// TIA Portal V20 export
TYPE "typeCmHmiInterfaceSoftCam"
// stored: Access Published, Namespace Unit1.Em4
   STRUCT
      sideTapeFixStageAxisX : "Unit1.Em4.typeCmHmiInterfaceSoftCamsideTapeFixStageAxisX";
      sideTapeFixStageAxisC : "Unit1.Em4.typeCmHmiInterfaceSoftCamsideTapeFixStageAxisC";
      sideTapeAttachmentAxisX : "Unit1.Em4.typeCmHmiInterfaceSoftCamsideTapeAttachmentAxisX";
      sideTapeAttachmentAxisY : "Unit1.Em4.typeCmHmiInterfaceSoftCamsideTapeAttachmentAxisY";
   END_STRUCT;
END_TYPE
